FUNCTION_BLOCK "ST10_Flow1_A1TableScan"
VAR_INPUT
  iSysInface : "RCS_SysComInterface_V1";
END_VAR
VAR_IN_OUT
  ioPM_Inface : "RCS_PMInterface_V1";
  ioStatus : Int;
END_VAR
VAR
  sCtrlMode : "SysFlowCtrlGraph";
  sUpdMES_Data : Bool;
  "工件放行中" : Bool;
  "前站站号" : UInt;
  "本站站号" : UInt;
  "弹窗Temp" : Array[1..10] of Int;
  AlarmID : Int;
  TON : Array[0..10] of TON_TIME;
  TOF : Array[0..10] of TOF_TIME;
  sUP : Array[0..10] of Bool;
  "更新RFID完成" : Bool;
  RT_DATA : G7_RTDataPlus_V6;
  Trans1 : G7_TransitionPlus_V6;
  Trans2 : G7_TransitionPlus_V6;
  Trans3 : G7_TransitionPlus_V6;
  Trans325 : G7_TransitionPlus_V6;
  Trans4 : G7_TransitionPlus_V6;
  Trans10 : G7_TransitionPlus_V6;
  Trans7 : G7_TransitionPlus_V6;
  Trans102 : G7_TransitionPlus_V6;
  Trans15 : G7_TransitionPlus_V6;
  Trans17 : G7_TransitionPlus_V6;
  Trans18 : G7_TransitionPlus_V6;
  Trans19 : G7_TransitionPlus_V6;
  Trans20 : G7_TransitionPlus_V6;
  Trans21 : G7_TransitionPlus_V6;
  Trans22 : G7_TransitionPlus_V6;
  Trans23 : G7_TransitionPlus_V6;
  Trans200 : G7_TransitionPlus_V6;
  "Fixture NG" : G7_TransitionPlus_V6;
  Trans767 : G7_TransitionPlus_V6;
  Trans768 : G7_TransitionPlus_V6;
  "Fixture OK" : G7_TransitionPlus_V6;
  Trans303 : G7_TransitionPlus_V6;
  Trans145 : G7_TransitionPlus_V6;
  Trans147 : G7_TransitionPlus_V6;
  Trans211 : G7_TransitionPlus_V6;
  Trans250 : G7_TransitionPlus_V6;
  Trans256 : G7_TransitionPlus_V6;
  Trans273 : G7_TransitionPlus_V6;
  ReadOK_2 : G7_TransitionPlus_V6;
  Trans254 : G7_TransitionPlus_V6;
  Trans278 : G7_TransitionPlus_V6;
  ReadNG_2 : G7_TransitionPlus_V6;
  ReadOK_1 : G7_TransitionPlus_V6;
  Trans279 : G7_TransitionPlus_V6;
  Trans282 : G7_TransitionPlus_V6;
  ReadNG_1 : G7_TransitionPlus_V6;
  Trans283 : G7_TransitionPlus_V6;
  Trans284 : G7_TransitionPlus_V6;
  Trans285 : G7_TransitionPlus_V6;
  ReadOK_3 : G7_TransitionPlus_V6;
  Trans286 : G7_TransitionPlus_V6;
  Trans287 : G7_TransitionPlus_V6;
  ReadNG_3 : G7_TransitionPlus_V6;
  Trans289 : G7_TransitionPlus_V6;
  Trans291 : G7_TransitionPlus_V6;
  ReadOK_4 : G7_TransitionPlus_V6;
  Trans292 : G7_TransitionPlus_V6;
  Trans293 : G7_TransitionPlus_V6;
  Trans294 : G7_TransitionPlus_V6;
  Trans295 : G7_TransitionPlus_V6;
  ReadNG_4 : G7_TransitionPlus_V6;
  ReadOK_5 : G7_TransitionPlus_V6;
  Trans296 : G7_TransitionPlus_V6;
  Trans297 : G7_TransitionPlus_V6;
  Trans298 : G7_TransitionPlus_V6;
  Trans315 : G7_TransitionPlus_V6;
  Trans299 : G7_TransitionPlus_V6;
  ReadNG_5 : G7_TransitionPlus_V6;
  ReadOK_6 : G7_TransitionPlus_V6;
  Trans300 : G7_TransitionPlus_V6;
  Trans301 : G7_TransitionPlus_V6;
  Trans302 : G7_TransitionPlus_V6;
  Trans304 : G7_TransitionPlus_V6;
  ReadNG_6 : G7_TransitionPlus_V6;
  ReadOK_7 : G7_TransitionPlus_V6;
  Trans305 : G7_TransitionPlus_V6;
  Trans306 : G7_TransitionPlus_V6;
  Trans235 : G7_TransitionPlus_V6;
  Trans307 : G7_TransitionPlus_V6;
  Trans308 : G7_TransitionPlus_V6;
  ReadNG_7 : G7_TransitionPlus_V6;
  Trans309 : G7_TransitionPlus_V6;
  ReadOK_8 : G7_TransitionPlus_V6;
  Trans310 : G7_TransitionPlus_V6;
  Trans311 : G7_TransitionPlus_V6;
  Trans312 : G7_TransitionPlus_V6;
  ReadNG_8 : G7_TransitionPlus_V6;
  Trans352 : G7_TransitionPlus_V6;
  Trans224 : G7_TransitionPlus_V6;
  Trans405 : G7_TransitionPlus_V6;
  Trans407 : G7_TransitionPlus_V6;
  Trans26 : G7_TransitionPlus_V6;
  "在线_1" : G7_TransitionPlus_V6;
  Trans408 : G7_TransitionPlus_V6;
  Trans27 : G7_TransitionPlus_V6;
  Trans229 : G7_TransitionPlus_V6;
  Trans268 : G7_TransitionPlus_V6;
  Trans270 : G7_TransitionPlus_V6;
  Trans271 : G7_TransitionPlus_V6;
  Trans274 : G7_TransitionPlus_V6;
  Trans624 : G7_TransitionPlus_V6;
  Trans605 : G7_TransitionPlus_V6;
  Trans420 : G7_TransitionPlus_V6;
  Trans255 : G7_TransitionPlus_V6;
  Trans288 : G7_TransitionPlus_V6;
  Trans619 : G7_TransitionPlus_V6;
  Trans622 : G7_TransitionPlus_V6;
  Trans623 : G7_TransitionPlus_V6;
  Trans280 : G7_TransitionPlus_V6;
  Trans281 : G7_TransitionPlus_V6;
  Trans419 : G7_TransitionPlus_V6;
  "离线_1" : G7_TransitionPlus_V6;
  Trans600 : G7_TransitionPlus_V6;
  Trans290 : G7_TransitionPlus_V6;
  Trans699 : G7_TransitionPlus_V6;
  Trans606 : G7_TransitionPlus_V6;
  Trans613 : G7_TransitionPlus_V6;
  Trans608 : G7_TransitionPlus_V6;
  Trans609 : G7_TransitionPlus_V6;
  Trans610 : G7_TransitionPlus_V6;
  Trans611 : G7_TransitionPlus_V6;
  Trans612 : G7_TransitionPlus_V6;
  Trans614 : G7_TransitionPlus_V6;
  Trans615 : G7_TransitionPlus_V6;
  Trans616 : G7_TransitionPlus_V6;
  Trans617 : G7_TransitionPlus_V6;
  F1_Initial : G7_StepPlus_V6;
  S2 : G7_StepPlus_V6;
  S3 : G7_StepPlus_V6;
  S4 : G7_StepPlus_V6;
  S5_MESInitial : G7_StepPlus_V6;
  "ServoReady?" : G7_StepPlus_V6;
  S8 : G7_StepPlus_V6;
  S9 : G7_StepPlus_V6;
  S10_InitialFinish : G7_StepPlus_V6;
  "Servo returns to2st Pos" : G7_StepPlus_V6;
  "Servo returns to1st Pos" : G7_StepPlus_V6;
  "Servo returns to3st Pos" : G7_StepPlus_V6;
  "Servo returns to4st Pos" : G7_StepPlus_V6;
  "Servo returns to3st Pos_1" : G7_StepPlus_V6;
  "Servo returns to3st Pos_2" : G7_StepPlus_V6;
  "Servo returns to3st Pos_3" : G7_StepPlus_V6;
  "Servo returns to3st Pos_4" : G7_StepPlus_V6;
  ProcessStart : G7_StepPlus_V6;
  "Determine TableFixtureStatus" : G7_StepPlus_V6;
  "A-Loading-01HorizontalCylinderToHP" : G7_StepPlus_V6;
  "A-Loading-01UpDownTakeCylinderToHP" : G7_StepPlus_V6;
  FixtureOK : G7_StepPlus_V6;
  Step128 : G7_StepPlus_V6;
  FixtureNG : G7_StepPlus_V6;
  "Tablecode reading" : G7_StepPlus_V6;
  ReadyReading : G7_StepPlus_V6;
  process : G7_StepPlus_V6;
  "Start 2st reading" : G7_StepPlus_V6;
  ReadNG1 : G7_StepPlus_V6;
  ReadNG2 : G7_StepPlus_V6;
  "Wait reading complete_" : G7_StepPlus_V6;
  DataMove_4 : G7_StepPlus_V6;
  DataMove_3 : G7_StepPlus_V6;
  "Check reader Ready2" : G7_StepPlus_V6;
  "Start 1st reading" : G7_StepPlus_V6;
  "Check reader Ready" : G7_StepPlus_V6;
  "Wait reading complete" : G7_StepPlus_V6;
  ReadNG3 : G7_StepPlus_V6;
  DataMove_5 : G7_StepPlus_V6;
  "Start 3st reading" : G7_StepPlus_V6;
  "Check reader Ready_4" : G7_StepPlus_V6;
  "Wait reading complete_4" : G7_StepPlus_V6;
  ReadNG4 : G7_StepPlus_V6;
  DataMove_6 : G7_StepPlus_V6;
  "Check reader Ready_5" : G7_StepPlus_V6;
  "Start 4st reading" : G7_StepPlus_V6;
  "Wait reading complete_5" : G7_StepPlus_V6;
  ReadNG7 : G7_StepPlus_V6;
  ReadNG5 : G7_StepPlus_V6;
  DataMove_7 : G7_StepPlus_V6;
  "Check reader Ready_6" : G7_StepPlus_V6;
  "Start 5st reading" : G7_StepPlus_V6;
  "Wait reading complete_6" : G7_StepPlus_V6;
  DataMove_1 : G7_StepPlus_V6;
  ReadNG6 : G7_StepPlus_V6;
  DataMove_8 : G7_StepPlus_V6;
  "Check reader Ready_7" : G7_StepPlus_V6;
  "Start 6st reading" : G7_StepPlus_V6;
  "Wait reading complete_7" : G7_StepPlus_V6;
  "Check reader Ready_8" : G7_StepPlus_V6;
  "Start 7st reading" : G7_StepPlus_V6;
  "Wait reading complete_9" : G7_StepPlus_V6;
  DataMove_2 : G7_StepPlus_V6;
  ReadNG8 : G7_StepPlus_V6;
  "Check reader Ready_9" : G7_StepPlus_V6;
  "Start 8st reading" : G7_StepPlus_V6;
  CodeCompare : G7_StepPlus_V6;
  "Wait reading complete_10" : G7_StepPlus_V6;
  Step262 : G7_StepPlus_V6;
  TableCodeReady : G7_StepPlus_V6;
  CodeCompareResult : G7_StepPlus_V6;
  "状态刷新100" : G7_StepPlus_V6;
  WaitChangeOverFinish : G7_StepPlus_V6;
  WaitReadyScanPrimit : G7_StepPlus_V6;
  WaitChangeOverStart : G7_StepPlus_V6;
  "Barcode mismatch" : G7_StepPlus_V6;
  WaitFixtureScanFinish : G7_StepPlus_V6;
  Step223 : G7_StepPlus_V6;
  Step400 : G7_StepPlus_V6;
  ProcessFinish : G7_StepPlus_V6;
  Step501 : G7_StepPlus_V6;
  "准备产品结果数据" : G7_StepPlus_V6;
  "是否在线1" : G7_StepPlus_V6;
  "MES保存开始" : G7_StepPlus_V6;
  "准备产品结果数据_1" : G7_StepPlus_V6;
  "复位MES保存命令" : G7_StepPlus_V6;
  "等待MES 保存Ready" : G7_StepPlus_V6;
  "505准备MES保存数据" : G7_StepPlus_V6;
  "置位MES保存命令" : G7_StepPlus_V6;
  "等待MES保存完成" : G7_StepPlus_V6;
  "MES保存完成" : G7_StepPlus_V6;
  "等待MES上传复位" : G7_StepPlus_V6;
  "MES保存结束" : G7_StepPlus_V6;
  Step617 : G7_StepPlus_V6;
  "状态刷新500" : G7_StepPlus_V6;
  "数据上传完成" : G7_StepPlus_V6;
  "MES上传复位超时" : G7_StepPlus_V6;
  "报警 MES保存超时" : G7_StepPlus_V6;
  "Process Finish" : G7_StepPlus_V6;
  ProcessFinsh : G7_StepPlus_V6;
END_VAR
VAR_TEMP
  Tempresult : USInt;
  "本站站号乘10" : UInt;
END_VAR
BEGIN
  // Původní jazyk: GRAPH
  // Zdroj XML: EXPORT/Program blocks/OP010/03_Auto/A1_TableLoad&Scan/ST10_Flow1_A1TableScan.xml
  // (Nebylo nalezeno StructuredText/FlgNet/StatementList; logika může být v GRAPH nebo v nepodporované reprezentaci.)
END_FUNCTION_BLOCK
